(* IEC 61131-3 sources: BOGDANKA/PLC, 4 files *)

(* ---- PLC_Typy_Danych.st ---- *)
(* ============================================================================
   BOGDANKA Szyb 2 - System Sterowania Nagrzewnicami
   Plik: PLC_Typy_Danych.st
   Opis: Definicje typów danych, struktur i enumeracji
   Standard: IEC 61131-3 Structured Text
   ============================================================================ *)

(* Typ wyliczeniowy: Scenariusze pracy *)
TYPE E_Scenariusz :
(
    S0 := 0,  // Brak ogrzewania
    S1 := 1,  // 1 nagrzewnica
    S2 := 2,  // 2 nagrzewnice
    S3 := 3,  // 3 nagrzewnice
    S4 := 4,  // 4 nagrzewnice
    S5 := 5,  // 5 nagrzewnic
    S6 := 6,  // 6 nagrzewnic
    S7 := 7,  // 7 nagrzewnic
    S8 := 8   // 8 nagrzewnic
);
END_TYPE

(* Typ wyliczeniowy: Układ pracy ciągów *)
TYPE E_Uklad :
(
    UKLAD_BRAK := 0,         // System wyłączony
    UKLAD_PODSTAWOWY := 1,   // C1 aktywny
    UKLAD_OGRANICZONY := 2   // C2 przez spinę
);
END_TYPE

(* Typ wyliczeniowy: Tryb pracy regulatora *)
TYPE E_TrybPracy :
(
    TRYB_MANUAL := 0,  // Sterowanie ręczne
    TRYB_AUTO := 1,    // Regulacja automatyczna PID
    TRYB_OFF := 2      // Wyłączony
);
END_TYPE

(* Typ wyliczeniowy: Stan nagrzewnicy *)
TYPE E_StanNagrzewnicy :
(
    STAN_OFF := 0,       // Wyłączona (zawór 20%)
    STAN_STARTING := 1,  // Uruchamianie
    STAN_RUNNING := 2,   // Praca normalna
    STAN_STOPPING := 3,  // Zatrzymywanie
    STAN_ERROR := 4      // Awaria
);
END_TYPE

(* Struktura: Dane nagrzewnicy *)
TYPE ST_Nagrzewnica :
STRUCT
    nNumer : USINT;                      // Numer nagrzewnicy (1-8)
    eStanNagrzewnicy : E_StanNagrzewnicy; // Aktualny stan
    fTemperaturaWylot : REAL;            // Temperatura na wylocie [°C]
    fPozycjaZaworu : REAL;               // Pozycja zaworu [%] (20-100)
    bPrzepustnicaDolotOtwarta : BOOL;    // Stan przepustnicy dolotowej
    bSprawna : BOOL;                     // Nagrzewnica sprawna
    bGotowoscOperacyjna : BOOL;          // Gotowość do pracy
    tCzasPracy : TIME;                   // Łączny czas pracy
    tCzasPostoju : TIME;                 // Łączny czas postoju
    dtTimestampZalaczenia : DT;          // Timestamp ostatniego załączenia
    dwLiczbaZalaczen : UDINT;            // Licznik załączeń
END_STRUCT
END_TYPE

(* Struktura: Dane wentylatora *)
TYPE ST_Wentylator :
STRUCT
    nNumer : USINT;                // Numer wentylatora (1-2)
    eTrybPracy : E_TrybPracy;      // Tryb: AUTO/MANUAL/OFF
    fCzestotliwosc : REAL;         // Częstotliwość [Hz] (25-50)
    fPradSilnika : REAL;           // Prąd silnika [A]
    bSprawny : BOOL;               // Wentylator sprawny
    bPracuje : BOOL;               // Wentylator w ruchu
    tCzasPracy : TIME;             // Łączny czas pracy
END_STRUCT
END_TYPE

(* Struktura: Parametry systemowe *)
TYPE ST_ParametrySystemowe :
STRUCT
    // Temperatury zadane
    fTzZadana : REAL := 50.0;         // Temperatura na wylocie nagrzewnicy [°C]
    fTsZadana : REAL := 2.0;          // Temperatura w szybie [°C]

    // Limity zaworu
    fPzMin : REAL := 20.0;            // Min. otwarcie zaworu [%]
    fPzMax : REAL := 100.0;           // Max. otwarcie zaworu [%]

    // Limity wentylatora
    fNWMin : REAL := 25.0;            // Min. częstotliwość [Hz]
    fNWMax : REAL := 50.0;            // Max. częstotliwość [Hz]

    // Parametry Algorytmu 5
    tCyklMonitoringuTemp : TIME := T#10s;       // Cykl odczytu temperatury
    tCzasUtrzymaniaPrzyAwarii : TIME := T#5m;   // Czas przy awarii czujnika
    nFiltrUsredniania : USINT := 3;             // Liczba próbek filtru
    tCzasStabilizacjiScenariusza : TIME := T#1m; // Min. czas w scenariuszu
    tCzasMiedzyZalaczeniami : TIME := T#30s;    // Odstęp między załączeniami
    tTimeoutZmianyScenariusza : TIME := T#10m;  // Timeout zmiany

    // Parametry Algorytmu 5A
    tOkresRotacjiUkladow : TIME := T#168h;      // Okres rotacji układów (7 dni)
    tHisterezaCzasowa : TIME := T#5m;           // Histereza czasowa
    tCyklPetliAlgorytmow : TIME := T#1m;        // Cykl pętli algorytmów

    // Parametry Algorytmu 5B
    tOkresRotacjiNagrzewnic : TIME := T#168h;   // Okres rotacji nagrzewnic
    tMinDeltaCzasu : TIME := T#1h;              // Min. różnica czasu dla rotacji
    tCzasStabilizacjiRotacji : TIME := T#30s;   // Czas stabilizacji po rotacji
END_STRUCT
END_TYPE

(* Struktura: Zmienne stanu systemu *)
TYPE ST_StanSystemu :
STRUCT
    // Temperatury
    fTZewn : REAL;                        // Temperatura zewnętrzna [°C]
    fTSzyb : REAL;                        // Temperatura w szybie [°C]
    bAlarmCzujnikTZewn : BOOL;            // Alarm awarii czujnika

    // Scenariusz
    eScenariuszAktualny : E_Scenariusz;   // Aktualny scenariusz
    eScenariuszWymagany : E_Scenariusz;   // Wymagany scenariusz
    dtTimestampOstatniejZmiany : DT;      // Timestamp ostatniej zmiany

    // Układ pracy
    eUkladAktualny : E_Uklad;             // Aktualny układ pracy
    tCzasPracyUkladuPodstawowego : TIME;  // Czas pracy układu podstawowego
    tCzasPracyUkladuOgraniczonego : TIME; // Czas pracy układu ograniczonego

    // Tryb pracy
    eTrybPracySystemu : E_TrybPracy;      // AUTO/MANUAL

    // Blokady koordynacji
    bZmianaUkladuWToku : BOOL;            // Blokada dla 5B
    bRotacjaNagrzewnicWToku : BOOL;       // Blokada dla 5A
    dtCzasOstatniejZmianyUkladu : DT;     // Dla koordynacji 5B
    dtCzasOstatniejRotacjiGlobalny : DT;  // Dla odstępu 15 min
END_STRUCT
END_TYPE

(* Struktura: Bufor pomiarów temperatury (filtr) *)
TYPE ST_BuforTemperatury :
STRUCT
    arWartosci : ARRAY[1..10] OF REAL;   // Bufor max 10 próbek
    nIndeks : USINT;                     // Aktualny indeks
    nLiczbaProbek : USINT;               // Liczba próbek w buforze
END_STRUCT
END_TYPE

(* Struktura: Statystyki rotacji *)
TYPE ST_StatystykiRotacji :
STRUCT
    dwLiczbaZmianUkladow : UDINT;        // Licznik rotacji układów
    dwLiczbaRotacjiNagrzewnic : UDINT;   // Licznik rotacji nagrzewnic
    tSredniCzasZmianyUkladu : TIME;      // Średni czas zmiany układu
    tSredniCzasRotacjiNagrzewnicy : TIME; // Średni czas rotacji
    fStosunEksploatacjiC1C2 : REAL;      // C1/C2 (cel: 1.0)
END_STRUCT
END_TYPE

(* ---- PLC_Algorytm_5_Wybor_Scenariusza.st ---- *)
(* ============================================================================
   BOGDANKA Szyb 2 - Algorytm 5: Automatyczny Wybór Scenariusza Pracy
   Plik: PLC_Algorytm_5_Wybor_Scenariusza.st
   Opis: Główny algorytm wyboru scenariusza na podstawie temperatury zewnętrznej
   Standard: IEC 61131-3 Structured Text
   ============================================================================ *)

PROGRAM PRG_Algorytm5_WyborScenariusza
VAR
    // Dane wejściowe
    Parametry : ST_ParametrySystemowe;
    StanSystemu : ST_StanSystemu;
    arrNagrzewnice : ARRAY[1..8] OF ST_Nagrzewnica;
    arrWentylatory : ARRAY[1..2] OF ST_Wentylator;

    // Zmienne lokalne
    BuforTZewn : ST_BuforTemperatury;
    fTZewnUsr : REAL;                        // Temperatura uśredniona
    fOstatniPoprawnyOdczyt : REAL := 20.0;  // Ostatni poprawny odczyt
    dtTimestampOstatniegoOdczytu : DT;

    // Timery
    tonCyklMonitoringu : TON;
    tonCzasStabilizacji : TON;

    // Zmienne pomocnicze
    bRotacjaMozliwa : BOOL;
    bRotacjaWymagana : BOOL;
    eScenariuszWymagany : E_Scenariusz;
    nWynik : INT;
END_VAR

(* ============================================================================
   GŁÓWNA PĘTLA - wykonywana cyklicznie
   ============================================================================ *)

// Timer cyklu monitoringu
tonCyklMonitoringu(IN := NOT tonCyklMonitoringu.Q, PT := Parametry.tCyklMonitoringuTemp);

IF tonCyklMonitoringu.Q THEN
    tonCyklMonitoringu(IN := FALSE);  // Reset timera

    // ========================================================================
    // KROK 1: Odczyt i walidacja temperatury zewnętrznej
    // ========================================================================

    IF (StanSystemu.fTZewn >= -40.0) AND (StanSystemu.fTZewn <= 50.0) THEN
        // Odczyt prawidłowy
        StanSystemu.bAlarmCzujnikTZewn := FALSE;
        fOstatniPoprawnyOdczyt := StanSystemu.fTZewn;
        dtTimestampOstatniegoOdczytu := DT_NOW();

        // Dodaj do bufora i oblicz średnią (filtr antyfluktuacyjny)
        BuforTZewn := FB_DodajDoBufora(BuforTZewn, StanSystemu.fTZewn, Parametry.nFiltrUsredniania);
        fTZewnUsr := FB_ObliczSrednia(BuforTZewn);
    ELSE
        // Awaria czujnika
        StanSystemu.bAlarmCzujnikTZewn := TRUE;

        IF (DT_NOW() - dtTimestampOstatniegoOdczytu) < Parametry.tCzasUtrzymaniaPrzyAwarii THEN
            // Utrzymaj ostatni scenariusz
            fTZewnUsr := fOstatniPoprawnyOdczyt;
        ELSE
            // Za długo bez odczytu - przełącz na tryb MANUAL
            StanSystemu.eTrybPracySystemu := TRYB_MANUAL;
            RETURN;  // Wyjdź z algorytmu
        END_IF;
    END_IF;

    // ========================================================================
    // KROK 2: Określ wymagany scenariusz na podstawie temperatury
    // ========================================================================

    eScenariuszWymagany := FB_OkreslScenariusz(fTZewnUsr, StanSystemu.eScenariuszAktualny);

    // ========================================================================
    // KROK 3: Sprawdź czy wymagana zmiana scenariusza
    // ========================================================================

    IF eScenariuszWymagany = StanSystemu.eScenariuszAktualny THEN
        RETURN;  // Brak zmiany - kontynuuj w aktualnym scenariuszu
    END_IF;

    // Sprawdź czas stabilizacji
    tonCzasStabilizacji(IN := TRUE, PT := Parametry.tCzasStabilizacjiScenariusza);

    IF NOT tonCzasStabilizacji.Q THEN
        RETURN;  // Za krótki czas od ostatniej zmiany
    END_IF;

    tonCzasStabilizacji(IN := FALSE);  // Reset timera

    // ========================================================================
    // KROK 4: Sprawdź tryb pracy
    // ========================================================================

    IF StanSystemu.eTrybPracySystemu <> TRYB_AUTO THEN
        RETURN;  // W trybie MANUAL operator kontroluje system
    END_IF;

    // ========================================================================
    // KROK 5: Wykonaj zmianę scenariusza
    // ========================================================================

    nWynik := FB_WykonajZmianeScenariusza(
        eScenariuszStary := StanSystemu.eScenariuszAktualny,
        eScenariuszNowy := eScenariuszWymagany,
        arrNagrzewnice := arrNagrzewnice,
        arrWentylatory := arrWentylatory,
        StanSystemu := StanSystemu,
        Parametry := Parametry
    );

    IF nWynik = 0 THEN
        // Sukces
        StanSystemu.eScenariuszAktualny := eScenariuszWymagany;
        StanSystemu.dtTimestampOstatniejZmiany := DT_NOW();
    ELSE
        // Błąd - pozostań w aktualnym scenariuszu
        // Alarm został już wygenerowany w funkcji
    END_IF;
END_IF;

END_PROGRAM

(* ============================================================================
   FUNKCJA: Określenie wymaganego scenariusza z histerezą
   ============================================================================ *)

FUNCTION FB_OkreslScenariusz : E_Scenariusz
VAR_INPUT
    fTZewn : REAL;                    // Temperatura zewnętrzna
    eAktualnyScenariusz : E_Scenariusz; // Aktualny scenariusz (dla histerezy)
END_VAR

    // Progi włączania (temperatura spada - dodajemy nagrzewnice)

    IF fTZewn >= 3.0 THEN
        FB_OkreslScenariusz := S0;
        RETURN;
    END_IF;

    // S1: -1°C < t ≤ 2°C (wyłączenie: t ≥ 3°C, histereza 1°C)
    IF fTZewn > 2.0 OR (fTZewn > -1.0 AND eAktualnyScenariusz = S0) THEN
        IF eAktualnyScenariusz = S0 THEN
            FB_OkreslScenariusz := S0;  // Zostań w S0
        ELSE
            FB_OkreslScenariusz := S1;  // Utrzymuj S1
        END_IF;
        RETURN;
    END_IF;

    IF fTZewn > -1.0 THEN
        FB_OkreslScenariusz := S1;
        RETURN;
    END_IF;

    // Histereza S1→S0
    IF fTZewn >= 0.0 AND eAktualnyScenariusz = S1 THEN
        FB_OkreslScenariusz := S0;
        RETURN;
    END_IF;

    // S2: -4°C < t ≤ -1°C (wyłączenie: t ≥ 0°C)
    IF fTZewn > -4.0 THEN
        FB_OkreslScenariusz := S2;
        RETURN;
    END_IF;

    IF fTZewn >= 0.0 AND eAktualnyScenariusz = S2 THEN
        FB_OkreslScenariusz := S1;
        RETURN;
    END_IF;

    // S3: -8°C < t ≤ -4°C (wyłączenie: t ≥ -3°C)
    IF fTZewn > -8.0 THEN
        FB_OkreslScenariusz := S3;
        RETURN;
    END_IF;

    IF fTZewn >= -3.0 AND eAktualnyScenariusz = S3 THEN
        FB_OkreslScenariusz := S2;
        RETURN;
    END_IF;

    // S4: -11°C < t ≤ -8°C (wyłączenie: t ≥ -6°C, histereza 2°C)
    IF fTZewn > -11.0 THEN
        FB_OkreslScenariusz := S4;
        RETURN;
    END_IF;

    IF fTZewn >= -6.0 AND eAktualnyScenariusz = S4 THEN
        FB_OkreslScenariusz := S3;
        RETURN;
    END_IF;

    // S5: -15°C < t ≤ -11°C (wyłączenie: t ≥ -10°C)
    IF fTZewn > -15.0 THEN
        FB_OkreslScenariusz := S5;
        RETURN;
    END_IF;

    IF fTZewn >= -10.0 AND eAktualnyScenariusz = S5 THEN
        FB_OkreslScenariusz := S4;
        RETURN;
    END_IF;

    // S6: -18°C < t ≤ -15°C (wyłączenie: t ≥ -13°C, histereza 2°C)
    IF fTZewn > -18.0 THEN
        FB_OkreslScenariusz := S6;
        RETURN;
    END_IF;

    IF fTZewn >= -13.0 AND eAktualnyScenariusz = S6 THEN
        FB_OkreslScenariusz := S5;
        RETURN;
    END_IF;

    // S7: -21°C < t ≤ -18°C (wyłączenie: t ≥ -15°C, histereza 3°C)
    IF fTZewn > -21.0 THEN
        FB_OkreslScenariusz := S7;
        RETURN;
    END_IF;

    IF fTZewn >= -15.0 AND eAktualnyScenariusz = S7 THEN
        FB_OkreslScenariusz := S6;
        RETURN;
    END_IF;

    // S8: t ≤ -21°C (wyłączenie: t ≥ -20°C)
    IF fTZewn <= -21.0 THEN
        FB_OkreslScenariusz := S8;
        RETURN;
    END_IF;

    IF fTZewn >= -20.0 AND eAktualnyScenariusz = S8 THEN
        FB_OkreslScenariusz := S7;
        RETURN;
    END_IF;

    // Domyślnie zwróć aktualny scenariusz
    FB_OkreslScenariusz := eAktualnyScenariusz;

END_FUNCTION

(* ============================================================================
   FUNKCJA: Wykonanie zmiany scenariusza
   Zwraca: 0 = sukces, -1 = błąd
   ============================================================================ *)

FUNCTION FB_WykonajZmianeScenariusza : INT
VAR_INPUT
    eScenariuszStary : E_Scenariusz;
    eScenariuszNowy : E_Scenariusz;
    arrNagrzewnice : ARRAY[1..8] OF ST_Nagrzewnica;
    arrWentylatory : ARRAY[1..2] OF ST_Wentylator;
    StanSystemu : ST_StanSystemu;
    Parametry : ST_ParametrySystemowe;
END_VAR
VAR
    dtStartZmiany : DT;
    nIloscStara : USINT;
    nIloscNowa : USINT;
    i : USINT;
    nWynik : INT;
END_VAR

    dtStartZmiany := DT_NOW();

    // Pobierz ilości nagrzewnic dla scenariuszy
    nIloscStara := FB_IloscNagrzewnicDlaScenariusza(eScenariuszStary);
    nIloscNowa := FB_IloscNagrzewnicDlaScenariusza(eScenariuszNowy);

    // ========================================================================
    // KROK 1: Zatrzymaj zbędne nagrzewnice (jeśli przechodzimy na niższy)
    // ========================================================================

    IF nIloscNowa < nIloscStara THEN
        FOR i := 1 TO (nIloscStara - nIloscNowa) DO
            // Pobierz nagrzewnicę do wyłączenia (najwyższy numer aktywny)
            nWynik := FB_WylaczNagrzewnice(arrNagrzewnice, 1);

            IF nWynik <> 0 THEN
                // Alarm już wygenerowany, ale kontynuuj
            END_IF;

            // Odstęp między wyłączeniami
            FB_Czekaj(Parametry.tCzasMiedzyZalaczeniami);
        END_FOR;
    END_IF;

    // ========================================================================
    // KROK 2: Skonfiguruj wentylatory
    // ========================================================================

    nWynik := FB_KonfigurujWentylatory(eScenariuszNowy, arrWentylatory, StanSystemu);

    IF nWynik <> 0 THEN
        FB_WykonajZmianeScenariusza := -1;
        RETURN;
    END_IF;

    FB_Czekaj(T#10s);  // Stabilizacja wentylatorów

    // ========================================================================
    // KROK 3: Skonfiguruj przepustnice
    // ========================================================================

    nWynik := FB_KonfigurujPrzepustnice(eScenariuszNowy, StanSystemu);

    IF nWynik <> 0 THEN
        FB_WykonajZmianeScenariusza := -1;
        RETURN;
    END_IF;

    FB_Czekaj(T#5s);

    // ========================================================================
    // KROK 4: Uruchom dodatkowe nagrzewnice (jeśli przechodzimy na wyższy)
    // ========================================================================

    IF nIloscNowa > nIloscStara THEN
        FOR i := 1 TO (nIloscNowa - nIloscStara) DO
            nWynik := FB_ZalaczNagrzewnice(arrNagrzewnice, eScenariuszNowy, StanSystemu);

            IF nWynik <> 0 THEN
                // Alarm, ale system może działać z mniejszą ilością
            END_IF;

            FB_Czekaj(Parametry.tCzasMiedzyZalaczeniami);
        END_FOR;
    END_IF;

    // ========================================================================
    // KROK 5: Weryfikacja
    // ========================================================================

    FB_Czekaj(T#30s);  // Czas na stabilizację

    IF FB_WeryfikujScenariusz(eScenariuszNowy, arrNagrzewnice, arrWentylatory) THEN
        FB_WykonajZmianeScenariusza := 0;  // Sukces
    ELSE
        FB_WykonajZmianeScenariusza := -1;  // Błąd weryfikacji
    END_IF;

END_FUNCTION

(* ---- PLC_Algorytm_5A_Rotacja_Ukladow.st ---- *)
(* ============================================================================
   BOGDANKA Szyb 2 - Algorytm 5A: Rotacja Układów Pracy Ciągów
   Plik: PLC_Algorytm_5A_Rotacja_Ukladow.st
   Opis: Cykliczna zmiana układów: Podstawowy ↔ Ograniczony
   Standard: IEC 61131-3 Structured Text
   ============================================================================ *)

PROGRAM PRG_Algorytm5A_RotacjaUkladow
VAR
    // Dane wejściowe
    Parametry : ST_ParametrySystemowe;
    StanSystemu : ST_StanSystemu;
    arrNagrzewnice : ARRAY[1..8] OF ST_Nagrzewnica;
    arrWentylatory : ARRAY[1..2] OF ST_Wentylator;

    // Zmienne lokalne
    dtCzasOstatniejZmianyUkladu : DT;
    bRotacjaMozliwa : BOOL;
    bRotacjaWymagana : BOOL;
    eNowyUklad : E_Uklad;

    // Timer
    tonCyklPetliAlgorytmu : TON;

    // Zmienne pomocnicze
    tCzasOdOstatniejZmiany : TIME;
    nWynik : INT;
END_VAR

(* ============================================================================
   GŁÓWNA PĘTLA - wykonywana cyklicznie
   ============================================================================ *)

// Timer cyklu algorytmu
tonCyklPetliAlgorytmu(IN := NOT tonCyklPetliAlgorytmu.Q, PT := Parametry.tCyklPetliAlgorytmow);

IF tonCyklPetliAlgorytmu.Q THEN
    tonCyklPetliAlgorytmu(IN := FALSE);  // Reset timera

    // ========================================================================
    // KROK 1: Sprawdź warunki rotacji
    // ========================================================================

    bRotacjaMozliwa := FALSE;

    // Rotacja tylko w scenariuszach S1-S4
    IF (StanSystemu.eScenariuszAktualny >= S1) AND
       (StanSystemu.eScenariuszAktualny <= S4) AND
       FB_WszystkieNagrzewniceC2Sprawne(arrNagrzewnice) AND
       arrWentylatory[2].bSprawny AND
       (StanSystemu.eTrybPracySystemu = TRYB_AUTO) THEN

        bRotacjaMozliwa := TRUE;
    ELSE
        // Rotacja niemożliwa - powrót do układu podstawowego jeśli był ograniczony
        IF StanSystemu.eUkladAktualny = UKLAD_OGRANICZONY THEN
            FB_WykonajZmianeUkladu(UKLAD_PODSTAWOWY, StanSystemu, arrNagrzewnice, arrWentylatory, Parametry);
        END_IF;

        RETURN;
    END_IF;

    // ========================================================================
    // KROK 2: Sprawdź czy upłynął okres rotacji
    // ========================================================================

    tCzasOdOstatniejZmiany := DT_NOW() - dtCzasOstatniejZmianyUkladu;

    IF tCzasOdOstatniejZmiany >= (Parametry.tOkresRotacjiUkladow - Parametry.tHisterezaCzasowa) THEN
        bRotacjaWymagana := TRUE;
    ELSE
        bRotacjaWymagana := FALSE;
        RETURN;
    END_IF;

    // ========================================================================
    // KROK 3: Określ nowy układ
    // ========================================================================

    IF StanSystemu.eUkladAktualny = UKLAD_PODSTAWOWY THEN
        eNowyUklad := UKLAD_OGRANICZONY;
    ELSE
        eNowyUklad := UKLAD_PODSTAWOWY;
    END_IF;

    // ========================================================================
    // KROK 4: Wykonaj zmianę układu
    // ========================================================================

    IF bRotacjaMozliwa AND bRotacjaWymagana THEN

        // Sprawdź czy Algorytm 5B nie wykonuje rotacji nagrzewnic
        IF StanSystemu.bRotacjaNagrzewnicWToku THEN
            // Zmiana odroczona
            RETURN;
        END_IF;

        // Ustaw blokadę dla Algorytmu 5B
        StanSystemu.bZmianaUkladuWToku := TRUE;

        // Wykonaj sekwencję zmiany układu
        nWynik := FB_WykonajZmianeUkladu(
            eDocelowyUklad := eNowyUklad,
            StanSystemu := StanSystemu,
            arrNagrzewnice := arrNagrzewnice,
            arrWentylatory := arrWentylatory,
            Parametry := Parametry
        );

        IF nWynik = 0 THEN
            // Sukces
            StanSystemu.eUkladAktualny := eNowyUklad;
            dtCzasOstatniejZmianyUkladu := DT_NOW();
            StanSystemu.dtCzasOstatniejZmianyUkladu := DT_NOW();  // Dla koordynacji z 5B
        END_IF;

        // Zwolnij blokadę
        StanSystemu.bZmianaUkladuWToku := FALSE;
    END_IF;

    // ========================================================================
    // KROK 5: Aktualizuj liczniki czasu pracy
    // ========================================================================

    IF StanSystemu.eUkladAktualny = UKLAD_PODSTAWOWY THEN
        StanSystemu.tCzasPracyUkladuPodstawowego := StanSystemu.tCzasPracyUkladuPodstawowego + Parametry.tCyklPetliAlgorytmow;
    ELSIF StanSystemu.eUkladAktualny = UKLAD_OGRANICZONY THEN
        StanSystemu.tCzasPracyUkladuOgraniczonego := StanSystemu.tCzasPracyUkladuOgraniczonego + Parametry.tCyklPetliAlgorytmow;
    END_IF;
END_IF;

END_PROGRAM

(* ============================================================================
   FUNKCJA: Wykonanie zmiany układu
   Zwraca: 0 = sukces, -1 = błąd
   ============================================================================ *)

FUNCTION FB_WykonajZmianeUkladu : INT
VAR_INPUT
    eDocelowyUklad : E_Uklad;
    StanSystemu : ST_StanSystemu;
    arrNagrzewnice : ARRAY[1..8] OF ST_Nagrzewnica;
    arrWentylatory : ARRAY[1..2] OF ST_Wentylator;
    Parametry : ST_ParametrySystemowe;
END_VAR
VAR
    i : USINT;
    nIloscAktywnych : USINT;
    nWymaganaIlosc : USINT;
END_VAR

    nWymaganaIlosc := FB_IloscNagrzewnicDlaScenariusza(StanSystemu.eScenariuszAktualny);

    IF eDocelowyUklad = UKLAD_OGRANICZONY THEN
        // ====================================================================
        // Przejście: Podstawowy → Ograniczony
        // ====================================================================

        // KROK 1: Zatrzymaj ciąg 1 (stopniowo)
        nIloscAktywnych := FB_LiczbaAktywnychNagrzewnicC1(arrNagrzewnice);

        FOR i := nIloscAktywnych TO 1 BY -1 DO
            FB_WylaczNagrzewnice(arrNagrzewnice, 1);  // Wyłącz z C1
            FB_Czekaj(T#30s);
        END_FOR;

        FB_ZatrzymajWentylator(arrWentylatory[1]);

        // KROK 2: Otwórz przepustnicę na spince ciągów
        FB_UstawPrzepustnice(PRZEPUSTNICA_SPINKA, TRUE);
        FB_Czekaj(T#10s);

        // KROK 3: Zamknij przepustnice ciągu 1
        FB_UstawPrzepustnice(PRZEPUSTNICA_KOLEKTOR_C1, FALSE);
        FB_UstawPrzepustnice(PRZEPUSTNICA_WYRZUTNIA_430, FALSE);

        // KROK 4: Uruchom ciąg 2 (stopniowo)
        FB_UruchomWentylator(arrWentylatory[2], 25.0);
        FB_Czekaj(T#10s);

        FOR i := 1 TO nWymaganaIlosc DO
            FB_ZalaczNagrzewnice(arrNagrzewnice, StanSystemu.eScenariuszAktualny, StanSystemu);
            FB_Czekaj(T#30s);
        END_FOR;

        // KROK 5: Aktywuj regulację PID dla W2
        FB_UstawWentylatorTryb(arrWentylatory[2], TRYB_AUTO);

    ELSE
        // ====================================================================
        // Przejście: Ograniczony → Podstawowy
        // ====================================================================

        // KROK 1: Zatrzymaj ciąg 2 (stopniowo)
        nIloscAktywnych := FB_LiczbaAktywnychNagrzewnicC2(arrNagrzewnice);

        FOR i := nIloscAktywnych TO 1 BY -1 DO
            FB_WylaczNagrzewnice(arrNagrzewnice, 2);  // Wyłącz z C2
            FB_Czekaj(T#30s);
        END_FOR;

        FB_ZatrzymajWentylator(arrWentylatory[2]);

        // KROK 2: Zamknij przepustnicę na spince ciągów
        FB_UstawPrzepustnice(PRZEPUSTNICA_SPINKA, FALSE);
        FB_Czekaj(T#10s);

        // KROK 3: Otwórz przepustnice ciągu 1
        FB_UstawPrzepustnice(PRZEPUSTNICA_KOLEKTOR_C1, TRUE);
        FB_UstawPrzepustnice(PRZEPUSTNICA_CIAG_C1, TRUE);
        FB_UstawPrzepustnice(PRZEPUSTNICA_WYRZUTNIA_430, TRUE);

        // KROK 4: Uruchom ciąg 1 (stopniowo)
        FB_UruchomWentylator(arrWentylatory[1], 25.0);
        FB_Czekaj(T#10s);

        FOR i := 1 TO nWymaganaIlosc DO
            FB_ZalaczNagrzewnice(arrNagrzewnice, StanSystemu.eScenariuszAktualny, StanSystemu);
            FB_Czekaj(T#30s);
        END_FOR;

        // KROK 5: Aktywuj regulację PID dla W1
        FB_UstawWentylatorTryb(arrWentylatory[1], TRYB_AUTO);
    END_IF;

    FB_WykonajZmianeUkladu := 0;  // Sukces

END_FUNCTION

(* ---- PLC_Algorytm_5B_Rotacja_Nagrzewnic.st ---- *)
(* ============================================================================
   BOGDANKA Szyb 2 - Algorytm 5B: Rotacja Nagrzewnic w Obrębie Ciągu
   Plik: PLC_Algorytm_5B_Rotacja_Nagrzewnic.st
   Opis: Cykliczna rotacja nagrzewnic - najdłużej pracująca → najdłużej w postoju
   Standard: IEC 61131-3 Structured Text
   ============================================================================ *)

PROGRAM PRG_Algorytm5B_RotacjaNagrzewnic
VAR
    // Dane wejściowe
    Parametry : ST_ParametrySystemowe;
    StanSystemu : ST_StanSystemu;
    arrNagrzewnice : ARRAY[1..8] OF ST_Nagrzewnica;
    arrWentylatory : ARRAY[1..2] OF ST_Wentylator;

    // Zmienne lokalne
    arrCzasOstatniejRotacji : ARRAY[1..2] OF DT;  // Dla każdego ciągu

    // Timer
    tonCyklPetliAlgorytmu : TON;

    // Zmienne pomocnicze
    nCiag : USINT;
    tCzasOdOstatniejRotacji : TIME;
    tCzasOdZmianyUkladu : TIME;
    tCzasOdOstatniejRotacjiGlobalnej : TIME;
    nIloscPracujacych : USINT;
    nIloscSprawnych : USINT;
    nNagrzewnicaDoWylaczenia : USINT;
    nNagrzewnicaDoZalaczenia : USINT;
    tMaxCzasPracy : TIME;
    tMaxCzasPostoju : TIME;
    tDeltaCzasu : TIME;
    nWynik : INT;
END_VAR

(* ============================================================================
   GŁÓWNA PĘTLA - wykonywana cyklicznie
   ============================================================================ *)

// Timer cyklu algorytmu
tonCyklPetliAlgorytmu(IN := NOT tonCyklPetliAlgorytmu.Q, PT := Parametry.tCyklPetliAlgorytmow);

IF tonCyklPetliAlgorytmu.Q THEN
    tonCyklPetliAlgorytmu(IN := FALSE);  // Reset timera

    // Przetwarzaj oba ciągi
    FOR nCiag := 1 TO 2 DO

        // ====================================================================
        // KROK 0: Sprawdź czy ciąg jest aktywny w aktualnym układzie/scenariuszu
        // ====================================================================

        // W S1-S4: tylko JEDEN ciąg aktywny (zależy od układu)
        IF (StanSystemu.eScenariuszAktualny >= S1) AND (StanSystemu.eScenariuszAktualny <= S4) THEN
            IF (StanSystemu.eUkladAktualny = UKLAD_PODSTAWOWY) AND (nCiag = 2) THEN
                CONTINUE;  // C2 wyłączony w układzie podstawowym
            END_IF;

            IF (StanSystemu.eUkladAktualny = UKLAD_OGRANICZONY) AND (nCiag = 1) THEN
                CONTINUE;  // C1 wyłączony w układzie ograniczonym
            END_IF;
        END_IF;

        // W S5-S8: C1 nie może rotować (brak rezerwowej - wszystkie 4 pracują)
        IF (StanSystemu.eScenariuszAktualny >= S5) AND (nCiag = 1) THEN
            CONTINUE;  // C1 rotacja niemożliwa
        END_IF;

        // ====================================================================
        // KROK 1: Aktualizuj liczniki czasu pracy i postoju
        // ====================================================================

        FB_AktualizujLicznikiCzasu(arrNagrzewnice, nCiag, Parametry.tCyklPetliAlgorytmow);

        // ====================================================================
        // KROK 2: Sprawdź warunki rotacji
        // ====================================================================

        // Koordynacja z Algorytmem 5A - sprawdź czy 5A nie wykonuje zmiany układu
        IF StanSystemu.bZmianaUkladuWToku THEN
            CONTINUE;  // Odrocz rotację
        END_IF;

        // Sprawdź czy upłynęła 1h od ostatniej zmiany układu (tylko S1-S4)
        IF (StanSystemu.eScenariuszAktualny >= S1) AND (StanSystemu.eScenariuszAktualny <= S4) THEN
            tCzasOdZmianyUkladu := DT_NOW() - StanSystemu.dtCzasOstatniejZmianyUkladu;
            IF tCzasOdZmianyUkladu < T#1h THEN
                CONTINUE;  // Za wcześnie po zmianie układu
            END_IF;
        END_IF;

        // Sprawdź odstęp 15 min od ostatniej rotacji (w dowolnym ciągu)
        tCzasOdOstatniejRotacjiGlobalnej := DT_NOW() - StanSystemu.dtCzasOstatniejRotacjiGlobalny;
        IF tCzasOdOstatniejRotacjiGlobalnej < T#15m THEN
            CONTINUE;  // Za krótki odstęp
        END_IF;

        // Sprawdź czy są nagrzewnice rezerwowe
        nIloscPracujacych := FB_LiczbaAktywnychNagrzewnic(arrNagrzewnice, nCiag);
        nIloscSprawnych := FB_LiczbaSprawnych(arrNagrzewnice, nCiag);

        IF nIloscSprawnych <= nIloscPracujacych THEN
            CONTINUE;  // Brak nagrzewnic rezerwowych
        END_IF;

        // Sprawdź czy upłynął okres rotacji
        tCzasOdOstatniejRotacji := DT_NOW() - arrCzasOstatniejRotacji[nCiag];

        IF tCzasOdOstatniejRotacji < Parametry.tOkresRotacjiNagrzewnic THEN
            CONTINUE;  // Nie upłynął jeszcze okres
        END_IF;

        // Sprawdź warunki stabilności
        IF NOT FB_WarunkiStabilnosciSpelnione(nCiag, arrWentylatory, StanSystemu) THEN
            CONTINUE;  // System niestabilny
        END_IF;

        // ====================================================================
        // KROK 3: Wybierz nagrzewnicę do wyłączenia i załączenia
        // ====================================================================

        // Znajdź nagrzewnicę najdłużej pracującą (aktywną)
        nNagrzewnicaDoWylaczenia := 0;
        tMaxCzasPracy := T#0s;

        nNagrzewnicaDoWylaczenia := FB_ZnajdzNajdluzejPracujaca(arrNagrzewnice, nCiag);

        IF nNagrzewnicaDoWylaczenia = 0 THEN
            CONTINUE;  // Nie znaleziono
        END_IF;

        tMaxCzasPracy := arrNagrzewnice[nNagrzewnicaDoWylaczenia].tCzasPracy;

        // Znajdź nagrzewnicę najdłużej w postoju (nieaktywną, sprawną)
        nNagrzewnicaDoZalaczenia := FB_ZnajdzNajdluzejWPostoju(arrNagrzewnice, nCiag);

        IF nNagrzewnicaDoZalaczenia = 0 THEN
            CONTINUE;  // Nie znaleziono
        END_IF;

        tMaxCzasPostoju := arrNagrzewnice[nNagrzewnicaDoZalaczenia].tCzasPostoju;

        // Sprawdź czy warto wykonać rotację
        tDeltaCzasu := tMaxCzasPracy - tMaxCzasPostoju;

        IF tDeltaCzasu < Parametry.tMinDeltaCzasu THEN
            CONTINUE;  // Różnica zbyt mała
        END_IF;

        // ====================================================================
        // KROK 4: Wykonaj rotację
        // ====================================================================

        // Ustaw blokadę dla Algorytmu 5A
        StanSystemu.bRotacjaNagrzewnicWToku := TRUE;

        nWynik := FB_WykonajRotacjeNagrzewnicy(
            nCiag := nCiag,
            nNStara := nNagrzewnicaDoWylaczenia,
            nNNowa := nNagrzewnicaDoZalaczenia,
            arrNagrzewnice := arrNagrzewnice,
            Parametry := Parametry
        );

        IF nWynik = 0 THEN
            // Sukces
            arrCzasOstatniejRotacji[nCiag] := DT_NOW();
            StanSystemu.dtCzasOstatniejRotacjiGlobalny := DT_NOW();
        END_IF;

        // Zwolnij blokadę
        StanSystemu.bRotacjaNagrzewnicWToku := FALSE;

    END_FOR;  // Koniec pętli ciągów
END_IF;

END_PROGRAM

(* ============================================================================
   FUNKCJA: Wykonanie rotacji nagrzewnicy
   Zwraca: 0 = sukces, -1 = błąd

   WAŻNA ZASADA BEZPIECZEŃSTWA:
   Najpierw ZAŁĄCZAMY nową nagrzewnicę, potem WYŁĄCZAMY starą
   ============================================================================ *)

FUNCTION FB_WykonajRotacjeNagrzewnicy : INT
VAR_INPUT
    nCiag : USINT;
    nNStara : USINT;
    nNNowa : USINT;
    arrNagrzewnice : ARRAY[1..8] OF ST_Nagrzewnica;
    Parametry : ST_ParametrySystemowe;
END_VAR
VAR
    fTempNNowa : REAL;
    fPozycjaZaworu : REAL;
    i : USINT;
END_VAR

    // ========================================================================
    // KROK 1: Przygotowanie nagrzewnicy nowej
    // ========================================================================

    IF NOT arrNagrzewnice[nNNowa].bGotowoscOperacyjna THEN
        FB_WykonajRotacjeNagrzewnicy := -1;
        RETURN;
    END_IF;

    // Ustaw zawór na pozycję startową (20%)
    FB_UstawZawor(arrNagrzewnice[nNNowa], Parametry.fPzMin);
    FB_Czekaj(T#5s);

    // ========================================================================
    // KROK 2: Załączenie nagrzewnicy nowej
    // ⚠️ W tym momencie pracuje: N_stara + N_nowa = WIĘCEJ niż wymaga scenariusz
    // To jest ZAMIERZONE dla bezpieczeństwa!
    // ========================================================================

    // Otwórz przepustnicę dolotową N_nowa
    FB_UstawPrzepustniceDolot(arrNagrzewnice[nNNowa], TRUE);
    FB_Czekaj(T#5s);

    // Otwórz zawór N_nowa stopniowo do 100%
    FOR fPozycjaZaworu := Parametry.fPzMin TO Parametry.fPzMax BY 10.0 DO
        FB_UstawZawor(arrNagrzewnice[nNNowa], fPozycjaZaworu);
        FB_Czekaj(T#2s);
    END_FOR;

    // Aktywuj regulator PID dla N_nowa
    FB_UstawRegulatorPID(arrNagrzewnice[nNNowa], TRYB_AUTO, Parametry.fTzZadana);
    FB_Czekaj(Parametry.tCzasStabilizacjiRotacji);

    // ========================================================================
    // KROK 3: Sprawdź stabilność temperatury
    // ========================================================================

    fTempNNowa := arrNagrzewnice[nNNowa].fTemperaturaWylot;

    IF ABS(fTempNNowa - Parametry.fTzZadana) > 5.0 THEN
        // Nowa nagrzewnica nie osiągnęła temperatury
        // Wycofaj zmianę - N_stara nadal pracuje, więc system bezpieczny
        FB_WylaczNagrzewnice(arrNagrzewnice, nCiag);
        FB_WykonajRotacjeNagrzewnicy := -1;
        RETURN;
    END_IF;

    // ========================================================================
    // KROK 4: Wyłączenie nagrzewnicy starej
    // ✅ Dopiero teraz, gdy mamy pewność że N_nowa działa, wyłączamy N_starą
    // Po tym kroku: poprawna ilość nagrzewnic zgodna ze scenariuszem
    // ========================================================================

    // Przełącz regulator PID dla N_stara w tryb MANUAL
    FB_UstawRegulatorPID(arrNagrzewnice[nNStara], TRYB_MANUAL, 0.0);

    // Zamknij zawór N_stara stopniowo do 20%
    fPozycjaZaworu := arrNagrzewnice[nNStara].fPozycjaZaworu;

    FOR i := 1 TO 10 DO
        fPozycjaZaworu := fPozycjaZaworu - 10.0;
        IF fPozycjaZaworu < Parametry.fPzMin THEN
            fPozycjaZaworu := Parametry.fPzMin;
        END_IF;
        FB_UstawZawor(arrNagrzewnice[nNStara], fPozycjaZaworu);
        FB_Czekaj(T#2s);
    END_FOR;

    // Poczekaj na stabilizację
    FB_Czekaj(Parametry.tCzasStabilizacjiRotacji);

    // Zamknij przepustnicę dolotową N_stara
    FB_UstawPrzepustniceDolot(arrNagrzewnice[nNStara], FALSE);

    // ========================================================================
    // KROK 5: Aktualizacja stanów
    // ========================================================================

    arrNagrzewnice[nNNowa].eStanNagrzewnicy := STAN_RUNNING;
    arrNagrzewnice[nNNowa].tCzasPostoju := T#0s;  // Zeruj licznik postoju
    arrNagrzewnice[nNNowa].dtTimestampZalaczenia := DT_NOW();

    arrNagrzewnice[nNStara].eStanNagrzewnicy := STAN_OFF;
    // Nie zeruj czasu pracy N_starej - pamiętamy łączny czas

    FB_WykonajRotacjeNagrzewnicy := 0;  // Sukces

END_FUNCTION
